FUNCTION_BLOCK FB_ReservoirTemperature
VAR_INPUT
	ReservoirVolume : REAL ; // L
	ReservoirHeaterIsOn : BOOL ;
	TotalPipeVolume : REAL ; // L
	CurrentPipeVolume : REAL ; // L
	TemperatureAfterGearbox : REAL ; //Celcius
END_VAR
VAR_OUTPUT
	ReservoirTemperature : REAL := Simulation_Parameters.AmbientTemperature ; //Celcius
END_VAR
VAR
	deltaTHeater : REAL := 0; // Celcius
	deltaTMixingGearboxReturn : REAL :=0 ; // Celcius
	
	ReservoirTemperatureNonFiltered : REAL := Simulation_Parameters.AmbientTemperature; // Celcius
	ReservoirConvectionHeat : REAL := 0 ; // Watt
	deltaTConvection : REAL := 0; // Celcius
	AmbientTemperature : REAL := Simulation_Parameters.AmbientTemperature; // Celcius
END_VAR

IF CurrentPipeVolume < (TotalPipeVolume) THEN
	deltaTMixingGearboxReturn := 0 ;
ELSE
	deltaTMixingGearboxReturn := f_deltaT_AfterMixingTwoFluids(	Mass1 := main.fb_MainLubeOilTemperatureAfterGearbox.PumpFlow,
																						SpecificHeatCapacity1 := simulation_parameters.SpecificHeatCapacityOil,
																						Temperature1 := TemperatureAfterGearbox,
																						Mass2 := ReservoirVolume,
																						SpecificHeatCapacity2 := simulation_parameters.SpecificHeatCapacityOil,
																						Temperature2 := ReservoirTemperature);
END_IF

	

IF ReservoirHeaterIsOn THEN
	deltaTHeater := f_CalculateDeltaT(	SpecificHeatCapacity := simulation_parameters.SpecificHeatCapacityOil,
										Density := Simulation_Parameters.OilDensity,
										Mass := ReservoirVolume,
										PowerInput := MainLubeoil_parameters.MainLubeOilReservoirHeaterPower);
ELSIF NOT ReservoirHeaterIsOn  THEN
	deltaTHeater := 0;
END_IF

ReservoirConvectionHeat := f_ReservoirConvectionHeat(ReservoirTemperature := ReservoirTemperature,
														AmbientTemperature := AmbientTemperature) ;
deltaTConvection := f_CalculateDeltaT (	SpecificHeatCapacity := simulation_parameters.SpecificHeatCapacityOil,
										Density := Simulation_Parameters.OilDensity,
										Mass := ReservoirVolume,
										PowerInput := ReservoirConvectionHeat);
										
ReservoirTemperatureNonFiltered := ReservoirTemperature + deltaTHeater + deltaTMixingGearboxReturn - deltaTConvection;
ReservoirTemperature := (1-simulation_parameters.TimeConstantReservoir)*ReservoirTemperature + simulation_parameters.TimeConstantReservoir*ReservoirTemperatureNonFiltered ;

END_FUNCTION_BLOCK

(* stored: Version 1.1.0.1, ProductVersion 3.1.4024.12
   POU FB_ReservoirTemperature: Id {e56d501c-cc3e-4275-8529-bf810e3f994f}, SpecialFunc None *)
